FUNCTION_BLOCK FB_Coordinador_SFC EXTENDS FB_Object_Template_SFC;
VAR_INPUT

//Discharger
	Discharger_Execute: BOOL;
	Discharger_Ready: BOOL;
	Discharger_Done: BOOL;
	Tray_1: BOOL;
	Tray_2: BOOL;
END_VAR
VAR_OUTPUT
	//Discharger
	Discharger_Ack: BOOL;

END_VAR
VAR
END_VAR

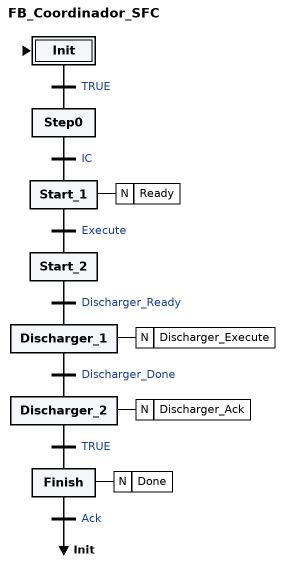
INITIAL_STEP Init:
END_STEP
TRANSITION FROM Init TO Step0
    := TRUE;
END_TRANSITION
STEP Step0:
END_STEP
TRANSITION FROM Step0 TO Start_1
    := IC;
END_TRANSITION
STEP Start_1:
    Ready(N);
END_STEP
TRANSITION FROM Start_1 TO Start_2
    := Execute;
END_TRANSITION
STEP Start_2:
END_STEP
TRANSITION FROM Start_2 TO Discharger_1
    := Discharger_Ready;
END_TRANSITION
STEP Discharger_1:
    Discharger_Execute(N);
END_STEP
TRANSITION FROM Discharger_1 TO Discharger_2
    := Discharger_Done;
END_TRANSITION
STEP Discharger_2:
    Discharger_Ack(N);
END_STEP
TRANSITION FROM Discharger_2 TO Finish
    := TRUE;
END_TRANSITION
STEP Finish:
    Done(N);
END_STEP
TRANSITION FROM Finish TO Init
    := Ack;
END_TRANSITION

END_FUNCTION_BLOCK

(* stored: Version 1.1.0.1, ProductVersion 3.1.4024.6
   POU FB_Coordinador_SFC: Id {16b6c9f6-6b37-46fb-9cbb-849c03f3e9f7}, SpecialFunc None *)
